Staubli VAL3: realTimeComm.pjx

--- realTimeComm.pjx ---
Parameters version=s7.9.1 stackSize=5000 millimeterUnit=true
Program file=arrayToJoint.pgx
Program file=Communication.pgx
Program file=jointToArray.pgx
Program file=moveTest.pgx
Program file=start.pgx
Program file=stop.pgx
Data file=realTimeComm.dtx

--- start.pgx ---
program start()
begin

  //测试开始
  call moveTest()


end

--- arrayToJoint.pgx ---
public program arrayToJoint(num& x_nNumInput[], jointRx& x_jJointOutput[])
  local num l_nNumOutput[6]
begin

  //==========解析两个机器人之间通讯收发的数据和指令==========

  //将数组数据解析成机器人的关节位置
  l_nNumOutput=x_nNumInput

  x_jJointOutput.j1=l_nNumOutput[0]
  x_jJointOutput.j2=l_nNumOutput[1]
  x_jJointOutput.j3=l_nNumOutput[2]
  x_jJointOutput.j4=l_nNumOutput[3]
  x_jJointOutput.j5=l_nNumOutput[4]
  x_jJointOutput.j6=l_nNumOutput[5]

end

--- moveTest.pgx ---
public program moveTest()
  local jointRx l_jJointRx_Me
  local jointRx l_jJointRx_Bro
begin

  l_jJointRx_Me={0,0,0,0,0,0}

  //测试机器人通讯
  while true

    movej(l_jJointRx_Me,flange,mNomSpeed)
    waitEndMove()
    delay(0.5)
    call Communication(l_jJointRx_Me,l_jJointRx_Bro)

    l_jJointRx_Me.j1=l_jJointRx_Me.j1+1
    l_jJointRx_Me.j2=l_jJointRx_Me.j2+1
    l_jJointRx_Me.j3=l_jJointRx_Me.j3+1
    l_jJointRx_Me.j4=l_jJointRx_Me.j4+1
    l_jJointRx_Me.j5=l_jJointRx_Me.j5+1
    l_jJointRx_Me.j6=l_jJointRx_Me.j6+1

  endWhile
end
